{attribute addProperty BoxType "EL2262-0000-0001"}
{attribute addProperty Id "CycCount0AT %Q*CycCount0_485675001620Sample0_0AT %Q*Sample_ABF5BEA9810GapAT %Q*EMPTY_STRUCTURE000CycCount1AT %Q*CycCount1_485675001620Sample1_0AT %Q*Sample_4351E8AC810Gap_1AT %Q*EMPTY_STRUCTURE000WcStateAT %I*WcState_64F6A8C6810InfoDataAT %I*InfoData_7231B2DD80100"}
{attribute addProperty CRC "2397240709"}
{attribute addProperty SizeInBites "136"}
{attribute addProperty SizeInBytes "17"}
TYPE EL2262_BE12C220 :
STRUCT
	{attribute addProperty Name "CycCount0"}
	CycCount0 : CycCount0_48567500;
	{attribute addProperty Name "Sample0_0"}
	Sample0_0 : Sample_ABF5BEA9;
	{attribute addProperty Name "Gap"}
	Gap : EMPTY_STRUCTURE;
	{attribute addProperty Name "CycCount1"}
	CycCount1 : CycCount1_48567500;
	{attribute addProperty Name "Sample1_0"}
	Sample1_0 : Sample_4351E8AC;
	{attribute addProperty Name "Gap_1"}
	Gap_1 : EMPTY_STRUCTURE;
	{attribute addProperty Name "WcState"}
	WcState : WcState_64F6A8C6;
	{attribute addProperty Name "InfoData"}
	InfoData : InfoData_7231B2DD;
END_STRUCT
END_TYPE

(* stored: Version 1.2.0.0, ProductVersion 3.1.4024.9
   DUT EL2262_BE12C220: Id {00c6bf6e-715d-48a6-9d11-d4065a6a1c83} *)
